FUNCTION_BLOCK Elevator EXTENDS A_Actuator
VAR_INPUT
END_VAR
VAR_OUTPUT
END_VAR
VAR
END_VAR

{warning 'Eigenschaftenimplementierung hinzufügen'}
PROPERTY cmd : E_ActuatorCmdType
GET
END_GET
SET
END_SET
END_PROPERTY

END_FUNCTION_BLOCK

(* stored: Version 1.1.0.1, ProductVersion 3.1.4024.2
   POU Elevator: Id {41bd1c28-57fc-4e4f-9823-dbd6c73872aa}, SpecialFunc None
   Property cmd: Id {bf01cc6c-3c44-4368-a27c-ea5a53013ace}
   Get Get: Id {0cf00c32-64b7-4a86-8be2-187f84f827f9}
   Set Set: Id {5e8b7a32-ca50-4e74-a7c4-9318f5fe3a31} *)
